(* Schneider Machine Expert - Basic project banda_asamblare_avioane, file version 2.6.0.0 *)
(* ProjectInformations: Name=New project *)

HARDWARE
  Cpu 0: TM221CE16R
  ModuleExtensionObject 0: TM3AM6/G
  EthernetConfiguration: NetworkName=M221, IpAllocationMode=FixedAddress, IpAddress=0.0.0.0, SubnetMask=0.0.0.0
  SerialLineConfiguration: Baud=Baud19200, Parity=ParityEven, DataBits=DataBits8, StopBits=StopBits1, PhysicalMedium=PhysicalMediumRs485, TransmissionMode=TransmissionModeModbusRtu, SlaveId=1, Addressing=SlaveAddressing
  MastTask: UsePeriodScanMode=false, PeriodScan=100
  FastTask: Period=255
  CpuBehavior: StartingMode=StartAsPreviousState, AutoSaveRamOnEeprom=true, WatchdogPeriod=250

SYMBOLS  (address, symbol, comment, settings)
  %IW0.0:X0 ARIPA_GEOMETRIE_VARIABILA
  %IW0.0:X1 ARIPA_TRIUNGIULARA
  %IW0.0:X2 ARIPA_TRAPEZOIDALA
  %IW0.0:X3 ARIPA_SAGEATA
  %IW0.0:X4 DISPOZITIV_ATERIZARE
  %IW0.0:X5 ELEROANE
  %IW0.0:X6 PROFUNDOR
  %IW0.0:X7 FLAPSURI
  %IW0.0:X8 VOLETI
  %IW0.0:X9 COMPENSATOARE
  %IW0.0:X10 FRANA_AERODINAMICA
  %IW0.0:X11 SISTEM_PROPULSIE
  %IW0.0:X12 SISTEM_HIDRAULIC
  %IW0.0:X13 SISTEME_CONTROL_ZBOR
  %IW0.0:X14 SISTEM_CONTROL_MOTOARE
  %IW0.0:X15 SISTEM_NAVIGATIE_AERIANA
  %IW0.1:X0 APARATURA_RADIO
  %IW0.1:X1 ARMAMENT_BORD
  %IW0.1:X2 BOMBARDAMENT_DIRIJARE_RACH
  %IW0.1:X3 BLINDAJ_PROTECTIE
  %IW0.1:X4 INSTALATIE_PNEUMATICA
  %IW0.1:X5 INSTALATIE_ELECTRICA
  %IW0.1:X6 INSTALATIE_ANTIGIVRAJ
  %M0       EXTERIOR_AVION_1
  %M1       FUZELAJUL_A_FOST_ALES
  %M2       ARIPA_PUSA
  %M3       ARIPA_CU_GEOM_VAR
  %M4       ARIPA_ADAUGATA
  %M5       AMPENAJE_ADAUGATE
  %M6       AMPENAJELE_AU_FOST_ADAUGATE
  %M7       ARIPA_TRIUNGH
  %M8       ARIPA_TRAPEZ
  %M9       ARIPA_SAG
  %M10      DISP_ATERIZARE_ADAUGAT
  %M11      ADAUGARE_DISP_ATERIZARE
  %M12      ADAUGARE_ELEROANE
  %M13      ADAUGARE_PROFUNDOR
  %M14      ADAUGARE_FLAPSURI
  %M15      ADAUGARE_VOLETI
  %M16      ADAUGARE_COMPENSATOARE
  %M17      ADAUGARE_FRANA
  %M18      ADAUGARE_SIS_PROP
  %M19      ADAUGARE_SIS_HIDRA
  %M20      ADAUGARE_SIS_CONTR_ZBOR
  %M21      ADAUGARE_SIS_CONTR_MOTOARE
  %M22      ADAUGARE_SIS_NAV
  %M23      ADAUGARE_RADIO
  %M24      ADAUGARE_ARMAMENT
  %M25      ARAGUARE_INSTALATIE_BOMB
  %M26      ADAUGARE_BLINDAJ
  %M27      ADAUGARE_INST_PNEUM
  %M28      ADAUGARE_INST_ELEC
  %M29      ADAUGARE_INST_ANTIGRIV
  %M30      SISTEM_1
  %M31      SISTEM_2
  %TM0      ADAUGARE_FUZELAJ  [Preset=3, Base=OneSecond]
  %TM1      ADAUGARE_ARIPI_AMPENAJE  [Preset=4, Base=OneSecond]
  %TM2        [Preset=7, Base=OneSecond]
  %TM3        [Preset=3, Base=OneSecond]
  %TM4        [Preset=4, Base=OneSecond]
  %TM5        [Preset=2, Base=OneSecond]
  %TM6        [Preset=3, Base=OneSecond]
  %TM7        [Preset=4, Base=OneSecond]
  %TM8        [Preset=2, Base=OneSecond]
  %C0       COUNTER_BOMBARDIER  [Preset=20]
  %C1       COUNTER_FIGHTER  [Preset=15]
  %C2       COUNTER_EXPLORER  [Preset=18]
  %I0.0     ASAMBLARE_AVION  "Asamblare_avion"
  %I0.1     BOMBARDIER
  %I0.2     FIGHTER
  %I0.3     EXPLORER
  %I0.4     ARIPA
  %I0.5     AMPENAJ_ORIZONTAL
  %I0.6     AMPENAJ_VERTICAL
  %I0.8     SENZOR_FOTOELECTRIC
  %Q0.0     EXTERIOR1
  %Q0.1     BOMBARDIER_FUZELAJ
  %Q0.2     FIGHTER_FUZELAJ
  %Q0.3     EXPLORER_FUZELAJ
  %Q0.4     ARIPA_GEOMETRIE_VAR
  %Q0.5     AVION
  %Q0.6     EXTERIOR
  %IW0.0      [Type=Type_0_10V, Scope=Scope_Normal, Minimum=0, Maximum=1000]
  %IW0.1      [Type=Type_0_10V, Scope=Scope_Normal, Minimum=0, Maximum=1000]
  %IW1.0      [Type=Type_4_20mA, Scope=Scope_Customized, Minimum=4000, Maximum=20000]
  %IW1.1      [Type=Type_4_20mA, Scope=Scope_Customized, Minimum=4000, Maximum=20000]

POU New POU
  (* SectionNumber=1 *)

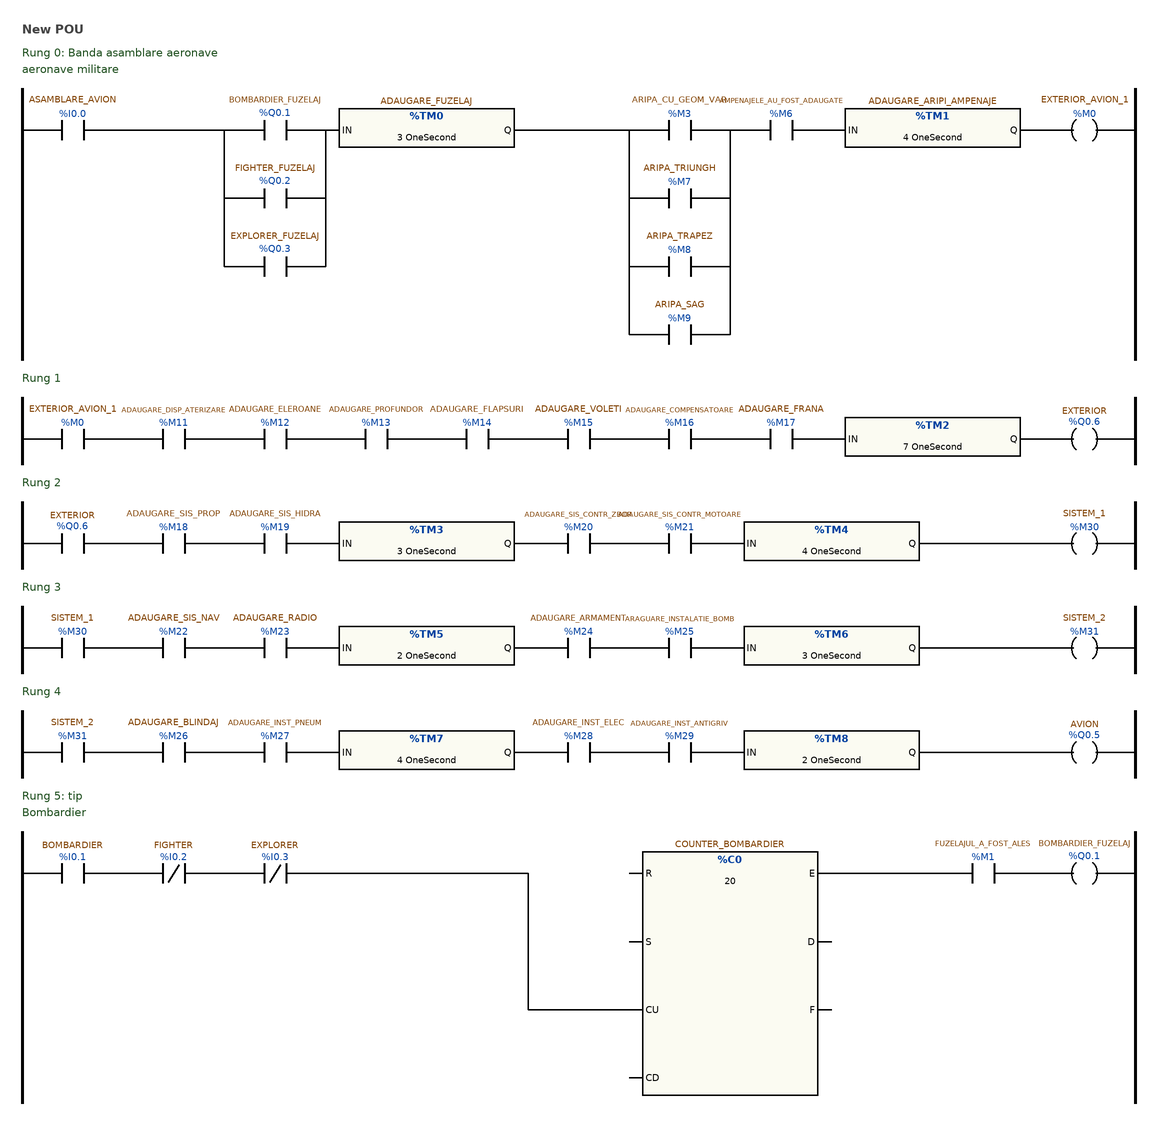

// Rung 0: Banda asamblare aeronave
// aeronave militare
  LD 1
  MULTIFB
  BLK %TM0                (* ADAUGARE_FUZELAJ *)
  LD 1
  AND %I0.0               (* ASAMBLARE_AVION *)
  AND( %Q0.1              (* BOMBARDIER_FUZELAJ *)
  OR %Q0.2                (* FIGHTER_FUZELAJ *)
  OR %Q0.3                (* EXPLORER_FUZELAJ *)
  )
  IN
  OUT_BLK
  LD Q
  ST %MW2009:X0
  END_BLK
  BLK %TM1                (* ADAUGARE_ARIPI_AMPENAJE *)
  LD %MW2009:X0
  AND( %M3                (* ARIPA_CU_GEOM_VAR *)
  OR %M7                  (* ARIPA_TRIUNGH *)
  OR %M8                  (* ARIPA_TRAPEZ *)
  OR %M9                  (* ARIPA_SAG *)
  )
  AND %M6                 (* AMPENAJELE_AU_FOST_ADAUGATE *)
  IN
  OUT_BLK
  LD Q
  ST %M0                  (* EXTERIOR_AVION_1 *)
  END_BLK
  MULTIFB
  // as ST:
  //   ADAUGARE_FUZELAJ(IN := ASAMBLARE_AVION AND (BOMBARDIER_FUZELAJ OR FIGHTER_FUZELAJ OR EXPLORER_FUZELAJ));
  //   ADAUGARE_ARIPI_AMPENAJE(IN := ADAUGARE_FUZELAJ.Q AND (ARIPA_CU_GEOM_VAR OR ARIPA_TRIUNGH OR ARIPA_TRAPEZ OR ARIPA_SAG) AND AMPENAJELE_AU_FOST_ADAUGATE);
  //   EXTERIOR_AVION_1 := ADAUGARE_ARIPI_AMPENAJE.Q;

// Rung 1
  BLK %TM2
  LD %M0                  (* EXTERIOR_AVION_1 *)
  AND %M11                (* ADAUGARE_DISP_ATERIZARE *)
  AND %M12                (* ADAUGARE_ELEROANE *)
  AND %M13                (* ADAUGARE_PROFUNDOR *)
  AND %M14                (* ADAUGARE_FLAPSURI *)
  AND %M15                (* ADAUGARE_VOLETI *)
  AND %M16                (* ADAUGARE_COMPENSATOARE *)
  AND %M17                (* ADAUGARE_FRANA *)
  IN
  OUT_BLK
  LD Q
  ST %Q0.6                (* EXTERIOR *)
  END_BLK
  // as ST:
  //   %TM2(IN := EXTERIOR_AVION_1 AND ADAUGARE_DISP_ATERIZARE AND ADAUGARE_ELEROANE AND ADAUGARE_PROFUNDOR AND ADAUGARE_FLAPSURI AND ADAUGARE_VOLETI AND ADAUGARE_COMPENSATOARE AND ADAUGARE_FRANA);
  //   EXTERIOR := %TM2.Q;

// Rung 2
  LD 1
  MULTIFB
  BLK %TM3
  LD 1
  AND %Q0.6               (* EXTERIOR *)
  AND %M18                (* ADAUGARE_SIS_PROP *)
  AND %M19                (* ADAUGARE_SIS_HIDRA *)
  IN
  OUT_BLK
  LD Q
  ST %MW2009:X0
  END_BLK
  BLK %TM4
  LD %MW2009:X0
  AND %M20                (* ADAUGARE_SIS_CONTR_ZBOR *)
  AND %M21                (* ADAUGARE_SIS_CONTR_MOTOARE *)
  IN
  OUT_BLK
  LD Q
  ST %M30                 (* SISTEM_1 *)
  END_BLK
  MULTIFB
  // as ST:
  //   %TM3(IN := EXTERIOR AND ADAUGARE_SIS_PROP AND ADAUGARE_SIS_HIDRA);
  //   %TM4(IN := %TM3.Q AND ADAUGARE_SIS_CONTR_ZBOR AND ADAUGARE_SIS_CONTR_MOTOARE);
  //   SISTEM_1 := %TM4.Q;

// Rung 3
  LD 1
  MULTIFB
  BLK %TM5
  LD 1
  AND %M30                (* SISTEM_1 *)
  AND %M22                (* ADAUGARE_SIS_NAV *)
  AND %M23                (* ADAUGARE_RADIO *)
  IN
  OUT_BLK
  LD Q
  ST %MW2009:X0
  END_BLK
  BLK %TM6
  LD %MW2009:X0
  AND %M24                (* ADAUGARE_ARMAMENT *)
  AND %M25                (* ARAGUARE_INSTALATIE_BOMB *)
  IN
  OUT_BLK
  LD Q
  ST %M31                 (* SISTEM_2 *)
  END_BLK
  MULTIFB
  // as ST:
  //   %TM5(IN := SISTEM_1 AND ADAUGARE_SIS_NAV AND ADAUGARE_RADIO);
  //   %TM6(IN := %TM5.Q AND ADAUGARE_ARMAMENT AND ARAGUARE_INSTALATIE_BOMB);
  //   SISTEM_2 := %TM6.Q;

// Rung 4
  LD 1
  MULTIFB
  BLK %TM7
  LD 1
  AND %M31                (* SISTEM_2 *)
  AND %M26                (* ADAUGARE_BLINDAJ *)
  AND %M27                (* ADAUGARE_INST_PNEUM *)
  IN
  OUT_BLK
  LD Q
  ST %MW2009:X0
  END_BLK
  BLK %TM8
  LD %MW2009:X0
  AND %M28                (* ADAUGARE_INST_ELEC *)
  AND %M29                (* ADAUGARE_INST_ANTIGRIV *)
  IN
  OUT_BLK
  LD Q
  ST %Q0.5                (* AVION *)
  END_BLK
  MULTIFB
  // as ST:
  //   %TM7(IN := SISTEM_2 AND ADAUGARE_BLINDAJ AND ADAUGARE_INST_PNEUM);
  //   %TM8(IN := %TM7.Q AND ADAUGARE_INST_ELEC AND ADAUGARE_INST_ANTIGRIV);
  //   AVION := %TM8.Q;

// Rung 5: tip
// Bombardier
  BLK %C0                 (* COUNTER_BOMBARDIER *)
  LD %I0.1                (* BOMBARDIER *)
  ANDN %I0.2              (* FIGHTER *)
  ANDN %I0.3              (* EXPLORER *)
  CU
  OUT_BLK
  LD E
  AND %M1                 (* FUZELAJUL_A_FOST_ALES *)
  ST %Q0.1                (* BOMBARDIER_FUZELAJ *)
  END_BLK
  // as ST:
  //   COUNTER_BOMBARDIER(CU := BOMBARDIER AND NOT FIGHTER AND NOT EXPLORER);
  //   BOMBARDIER_FUZELAJ := COUNTER_BOMBARDIER.E AND FUZELAJUL_A_FOST_ALES;

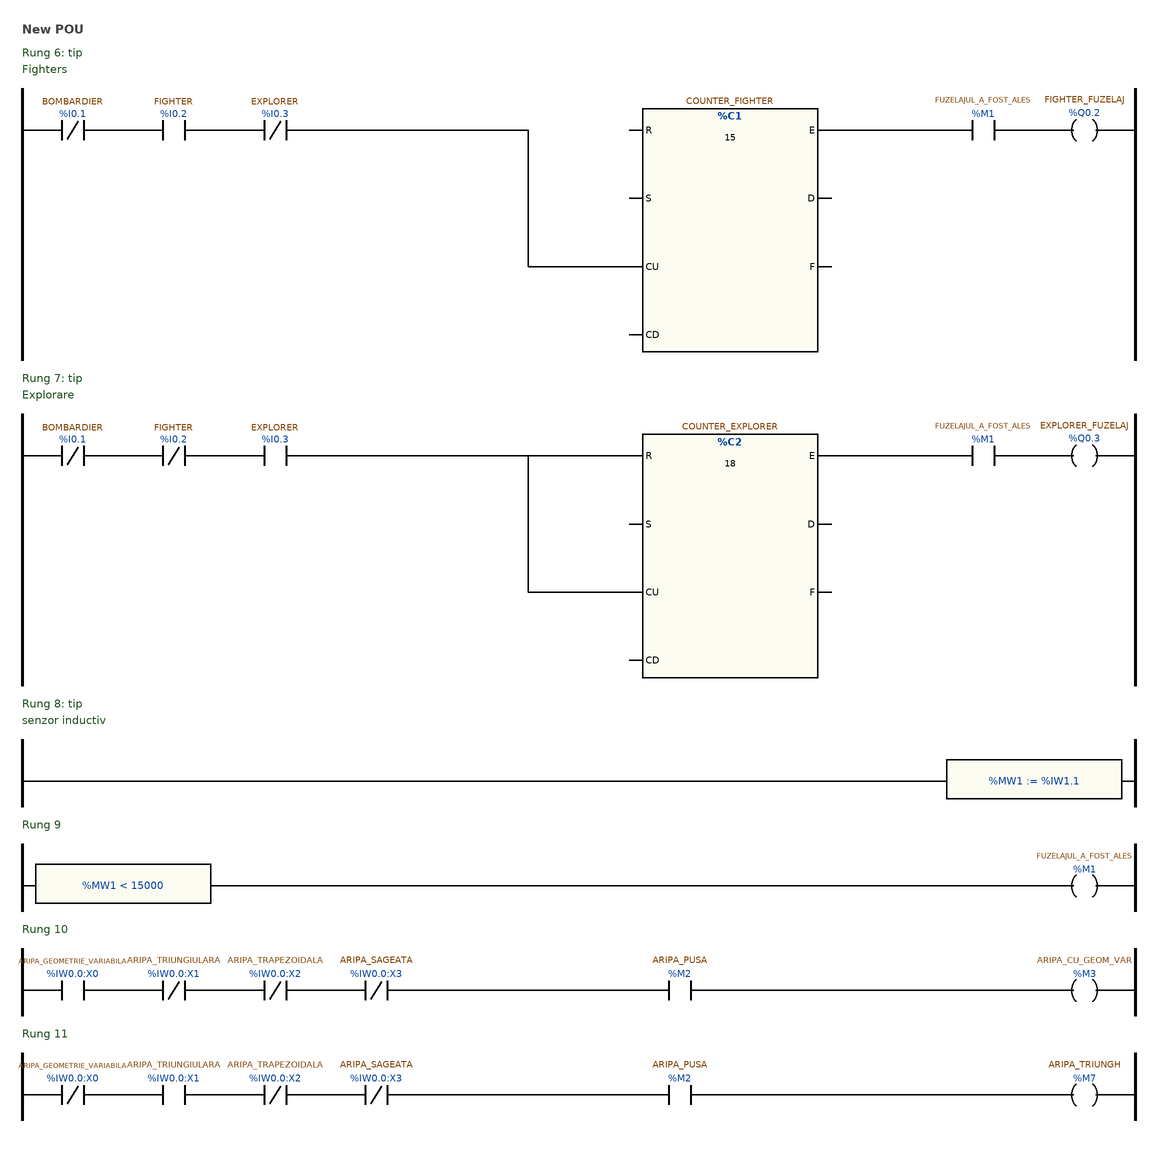

// Rung 6: tip
// Fighters
  BLK %C1                 (* COUNTER_FIGHTER *)
  LDN %I0.1               (* BOMBARDIER *)
  AND %I0.2               (* FIGHTER *)
  ANDN %I0.3              (* EXPLORER *)
  CU
  OUT_BLK
  LD E
  AND %M1                 (* FUZELAJUL_A_FOST_ALES *)
  ST %Q0.2                (* FIGHTER_FUZELAJ *)
  END_BLK
  // as ST:
  //   COUNTER_FIGHTER(CU := NOT BOMBARDIER AND FIGHTER AND NOT EXPLORER);
  //   FIGHTER_FUZELAJ := COUNTER_FIGHTER.E AND FUZELAJUL_A_FOST_ALES;

// Rung 7: tip
// Explorare
  BLK %C2                 (* COUNTER_EXPLORER *)
  LDN %I0.1               (* BOMBARDIER *)
  ANDN %I0.2              (* FIGHTER *)
  AND %I0.3               (* EXPLORER *)
  R
  CU
  OUT_BLK
  LD E
  AND %M1                 (* FUZELAJUL_A_FOST_ALES *)
  ST %Q0.3                (* EXPLORER_FUZELAJ *)
  END_BLK
  // as ST:
  //   COUNTER_EXPLORER(R := NOT BOMBARDIER AND NOT FIGHTER AND EXPLORER, CU := NOT BOMBARDIER AND NOT FIGHTER AND EXPLORER);
  //   EXPLORER_FUZELAJ := COUNTER_EXPLORER.E AND FUZELAJUL_A_FOST_ALES;

// Rung 8: tip
// senzor inductiv
  LD 1
  [ %MW1 := %IW1.1 ]
  // as ST:
  //   %MW1 := %IW1.1;

// Rung 9
  LD [ %MW1 < 15000 ]
  ST %M1                  (* FUZELAJUL_A_FOST_ALES *)
  // as ST:
  //   FUZELAJUL_A_FOST_ALES := %MW1 < 15000;

// Rung 10
  LD %IW0.0:X0
  ANDN %IW0.0:X1
  ANDN %IW0.0:X2
  ANDN %IW0.0:X3
  AND %M2                 (* ARIPA_PUSA *)
  ST %M3                  (* ARIPA_CU_GEOM_VAR *)
  // as ST:
  //   ARIPA_CU_GEOM_VAR := %IW0.0:X0 AND NOT %IW0.0:X1 AND NOT %IW0.0:X2 AND NOT %IW0.0:X3 AND ARIPA_PUSA;

// Rung 11
  LDN %IW0.0:X0
  AND %IW0.0:X1
  ANDN %IW0.0:X2
  ANDN %IW0.0:X3
  AND %M2                 (* ARIPA_PUSA *)
  ST %M7                  (* ARIPA_TRIUNGH *)
  // as ST:
  //   ARIPA_TRIUNGH := NOT %IW0.0:X0 AND %IW0.0:X1 AND NOT %IW0.0:X2 AND NOT %IW0.0:X3 AND ARIPA_PUSA;

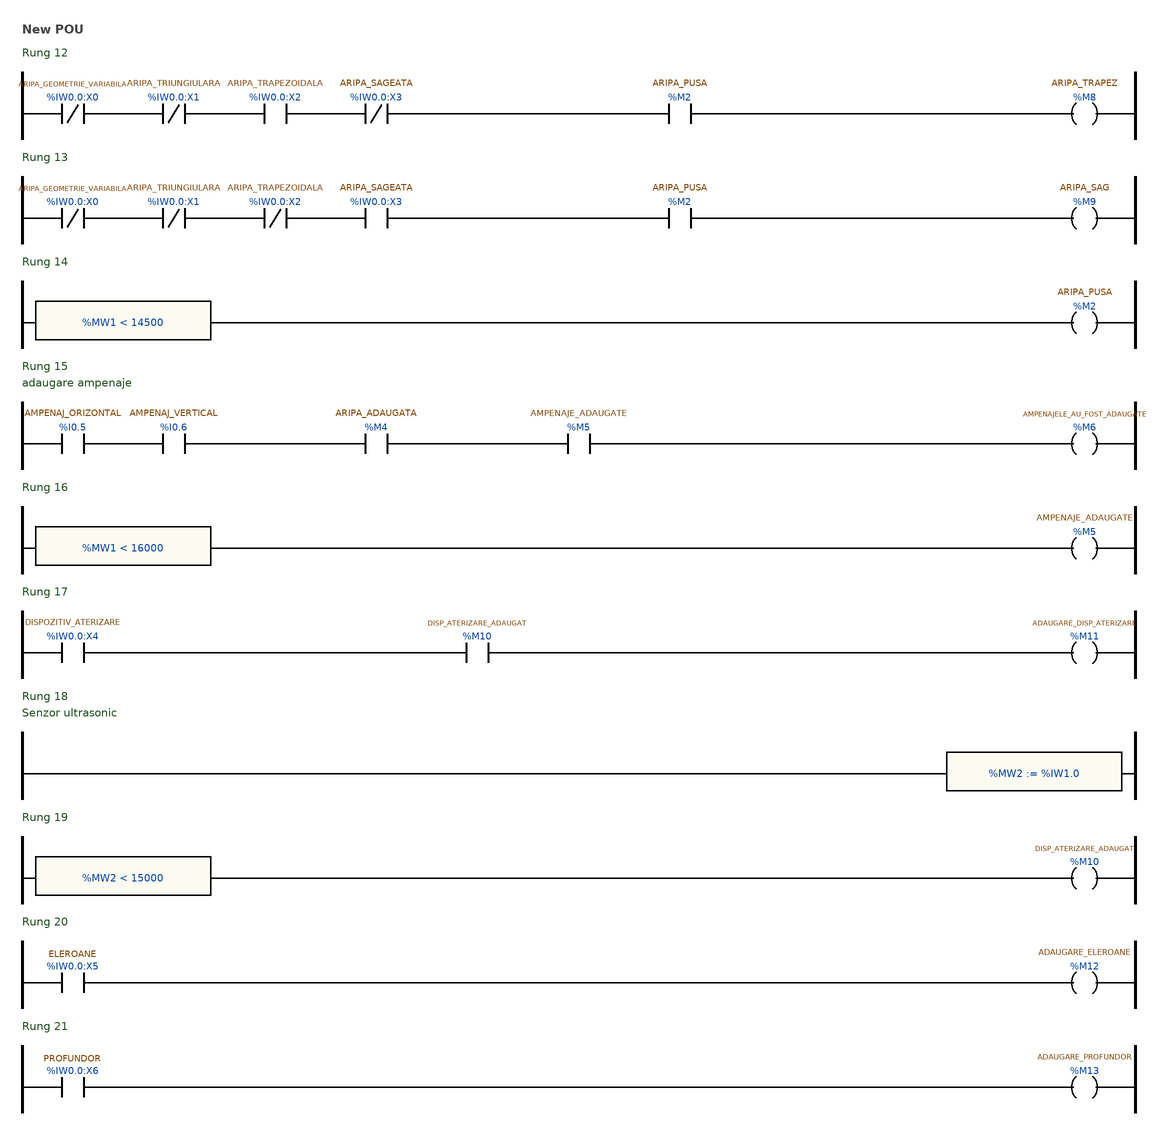

// Rung 12
  LDN %IW0.0:X0
  ANDN %IW0.0:X1
  AND %IW0.0:X2
  ANDN %IW0.0:X3
  AND %M2                 (* ARIPA_PUSA *)
  ST %M8                  (* ARIPA_TRAPEZ *)
  // as ST:
  //   ARIPA_TRAPEZ := NOT %IW0.0:X0 AND NOT %IW0.0:X1 AND %IW0.0:X2 AND NOT %IW0.0:X3 AND ARIPA_PUSA;

// Rung 13
  LDN %IW0.0:X0
  ANDN %IW0.0:X1
  ANDN %IW0.0:X2
  AND %IW0.0:X3
  AND %M2                 (* ARIPA_PUSA *)
  ST %M9                  (* ARIPA_SAG *)
  // as ST:
  //   ARIPA_SAG := NOT %IW0.0:X0 AND NOT %IW0.0:X1 AND NOT %IW0.0:X2 AND %IW0.0:X3 AND ARIPA_PUSA;

// Rung 14
  LD [ %MW1 < 14500 ]
  ST %M2                  (* ARIPA_PUSA *)
  // as ST:
  //   ARIPA_PUSA := %MW1 < 14500;

// Rung 15
// adaugare ampenaje
  LD %I0.5                (* AMPENAJ_ORIZONTAL *)
  AND %I0.6               (* AMPENAJ_VERTICAL *)
  AND %M4                 (* ARIPA_ADAUGATA *)
  AND %M5                 (* AMPENAJE_ADAUGATE *)
  ST %M6                  (* AMPENAJELE_AU_FOST_ADAUGATE *)
  // as ST:
  //   AMPENAJELE_AU_FOST_ADAUGATE := AMPENAJ_ORIZONTAL AND AMPENAJ_VERTICAL AND ARIPA_ADAUGATA AND AMPENAJE_ADAUGATE;

// Rung 16
  LD [ %MW1 < 16000 ]
  ST %M5                  (* AMPENAJE_ADAUGATE *)
  // as ST:
  //   AMPENAJE_ADAUGATE := %MW1 < 16000;

// Rung 17
  LD %IW0.0:X4
  AND %M10                (* DISP_ATERIZARE_ADAUGAT *)
  ST %M11                 (* ADAUGARE_DISP_ATERIZARE *)
  // as ST:
  //   ADAUGARE_DISP_ATERIZARE := %IW0.0:X4 AND DISP_ATERIZARE_ADAUGAT;

// Rung 18
// Senzor ultrasonic
  LD 1
  [ %MW2 := %IW1.0 ]
  // as ST:
  //   %MW2 := %IW1.0;

// Rung 19
  LD [ %MW2 < 15000 ]
  ST %M10                 (* DISP_ATERIZARE_ADAUGAT *)
  // as ST:
  //   DISP_ATERIZARE_ADAUGAT := %MW2 < 15000;

// Rung 20
  LD %IW0.0:X5
  ST %M12                 (* ADAUGARE_ELEROANE *)
  // as ST:
  //   ADAUGARE_ELEROANE := %IW0.0:X5;

// Rung 21
  LD %IW0.0:X6
  ST %M13                 (* ADAUGARE_PROFUNDOR *)
  // as ST:
  //   ADAUGARE_PROFUNDOR := %IW0.0:X6;

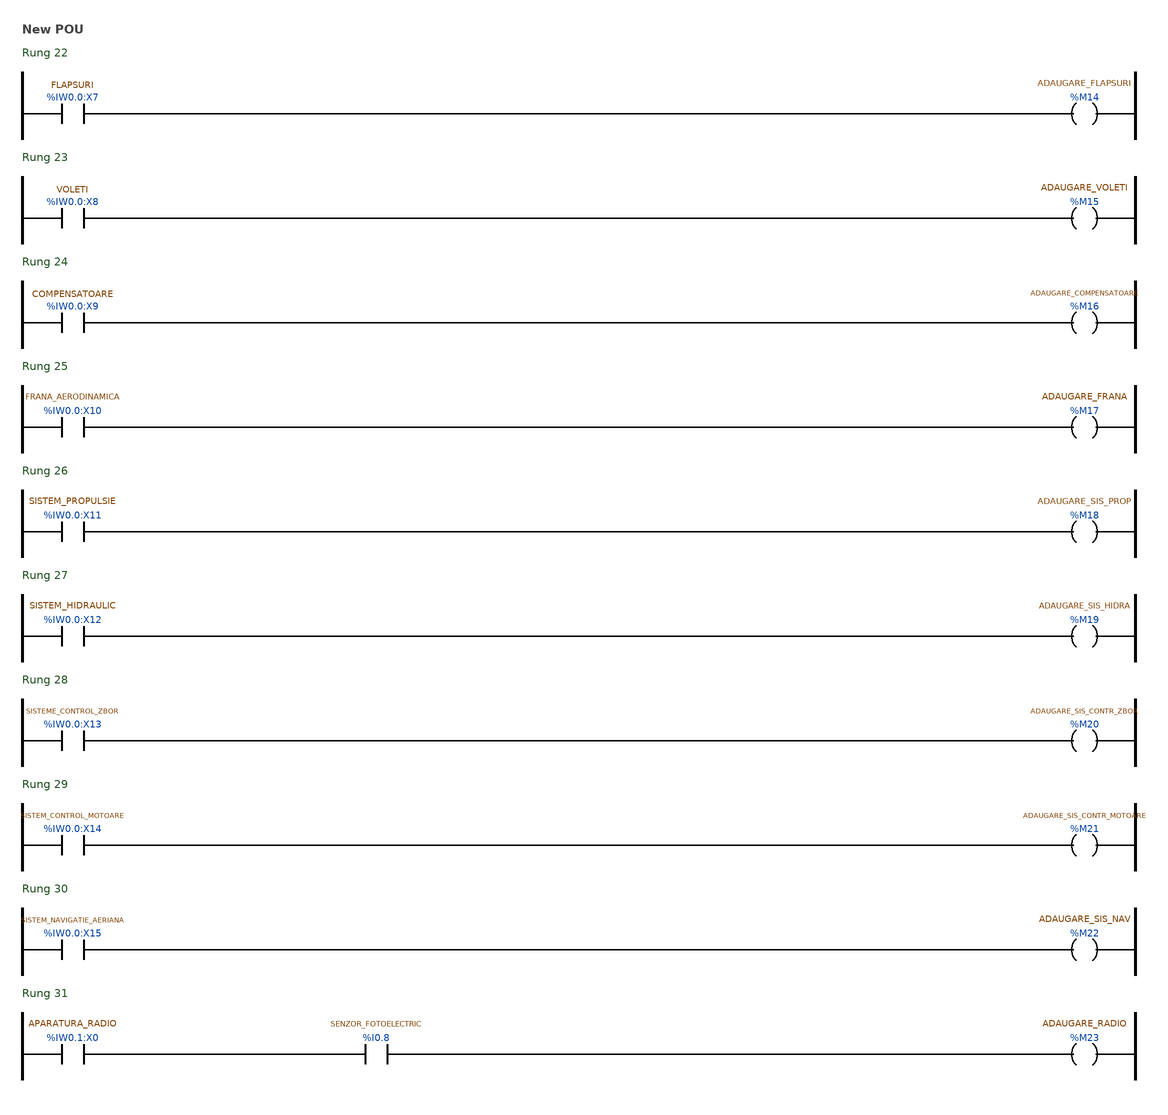

// Rung 22
  LD %IW0.0:X7
  ST %M14                 (* ADAUGARE_FLAPSURI *)
  // as ST:
  //   ADAUGARE_FLAPSURI := %IW0.0:X7;

// Rung 23
  LD %IW0.0:X8
  ST %M15                 (* ADAUGARE_VOLETI *)
  // as ST:
  //   ADAUGARE_VOLETI := %IW0.0:X8;

// Rung 24
  LD %IW0.0:X9
  ST %M16                 (* ADAUGARE_COMPENSATOARE *)
  // as ST:
  //   ADAUGARE_COMPENSATOARE := %IW0.0:X9;

// Rung 25
  LD %IW0.0:X10
  ST %M17                 (* ADAUGARE_FRANA *)
  // as ST:
  //   ADAUGARE_FRANA := %IW0.0:X10;

// Rung 26
  LD %IW0.0:X11
  ST %M18                 (* ADAUGARE_SIS_PROP *)
  // as ST:
  //   ADAUGARE_SIS_PROP := %IW0.0:X11;

// Rung 27
  LD %IW0.0:X12
  ST %M19                 (* ADAUGARE_SIS_HIDRA *)
  // as ST:
  //   ADAUGARE_SIS_HIDRA := %IW0.0:X12;

// Rung 28
  LD %IW0.0:X13
  ST %M20                 (* ADAUGARE_SIS_CONTR_ZBOR *)
  // as ST:
  //   ADAUGARE_SIS_CONTR_ZBOR := %IW0.0:X13;

// Rung 29
  LD %IW0.0:X14
  ST %M21                 (* ADAUGARE_SIS_CONTR_MOTOARE *)
  // as ST:
  //   ADAUGARE_SIS_CONTR_MOTOARE := %IW0.0:X14;

// Rung 30
  LD %IW0.0:X15
  ST %M22                 (* ADAUGARE_SIS_NAV *)
  // as ST:
  //   ADAUGARE_SIS_NAV := %IW0.0:X15;

// Rung 31
  LD %IW0.1:X0
  AND %I0.8               (* SENZOR_FOTOELECTRIC *)
  ST %M23                 (* ADAUGARE_RADIO *)
  // as ST:
  //   ADAUGARE_RADIO := %IW0.1:X0 AND SENZOR_FOTOELECTRIC;

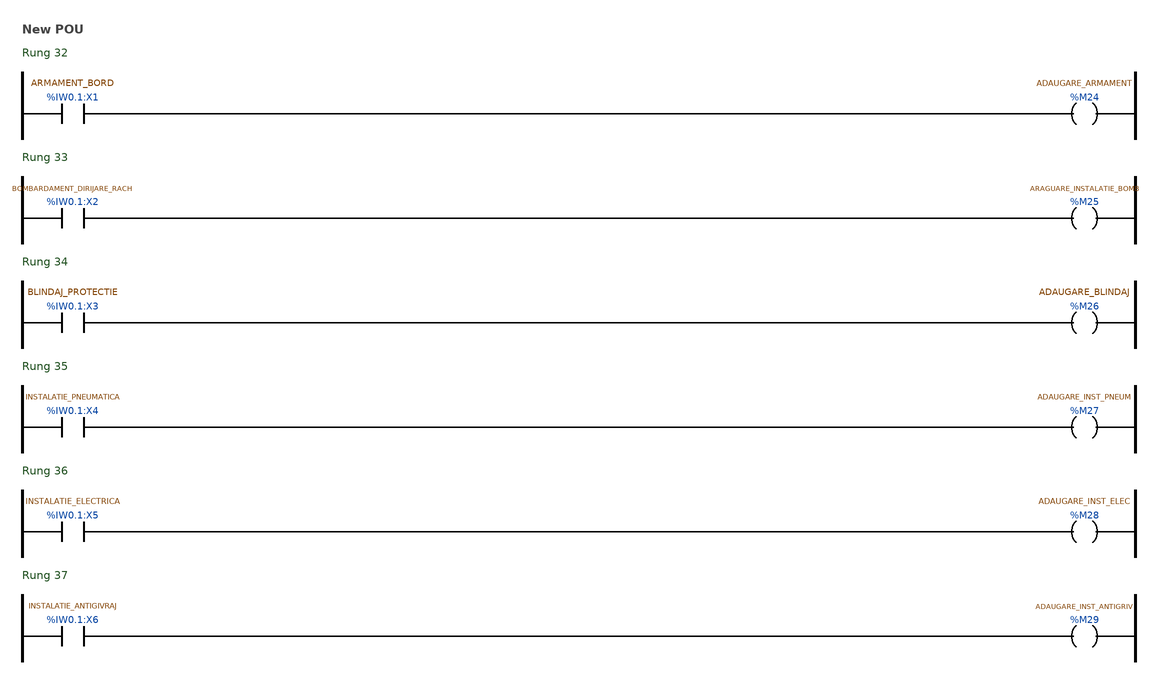

// Rung 32
  LD %IW0.1:X1
  ST %M24                 (* ADAUGARE_ARMAMENT *)
  // as ST:
  //   ADAUGARE_ARMAMENT := %IW0.1:X1;

// Rung 33
  LD %IW0.1:X2
  ST %M25                 (* ARAGUARE_INSTALATIE_BOMB *)
  // as ST:
  //   ARAGUARE_INSTALATIE_BOMB := %IW0.1:X2;

// Rung 34
  LD %IW0.1:X3
  ST %M26                 (* ADAUGARE_BLINDAJ *)
  // as ST:
  //   ADAUGARE_BLINDAJ := %IW0.1:X3;

// Rung 35
  LD %IW0.1:X4
  ST %M27                 (* ADAUGARE_INST_PNEUM *)
  // as ST:
  //   ADAUGARE_INST_PNEUM := %IW0.1:X4;

// Rung 36
  LD %IW0.1:X5
  ST %M28                 (* ADAUGARE_INST_ELEC *)
  // as ST:
  //   ADAUGARE_INST_ELEC := %IW0.1:X5;

// Rung 37
  LD %IW0.1:X6
  ST %M29                 (* ADAUGARE_INST_ANTIGRIV *)
  // as ST:
  //   ADAUGARE_INST_ANTIGRIV := %IW0.1:X6;
